// TIA Portal V16 export
// export: Created 2021-07-21T13:08:43.8324365Z, ExportSetting WithDefaults, DisplayName Totally Integrated Automation Portal, DisplayVersion V16 Update 3, DisplayName TIA Portal Version Control Interface, DisplayVersion V16 Update 2, DisplayName TIA Portal Openness, DisplayVersion V16 Update 3, DisplayName STEP 7 Professional, DisplayVersion V16 Update 3, DisplayName STEP 7 Safety, DisplayVersion V16, DisplayName WinCC Professional, DisplayVersion V16 Update 3
TYPE "UT31001_Dy_DevValveIsol"
TITLE = Dynamic UDT [Instrumentation] — Analog Instrument Read, Scale and Monitor
// Analogue Instrument Read and Scale
// stored: IsFailsafeCompliant false
   STRUCT
      revInfo : "UT01000_St_SysRevision";   // Revision information
      ___________0010_0 { ExternalAccessible := 'False'; ExternalVisible := 'False'; ExternalWritable := 'False'} : Int;
      ___________0010_1 { ExternalAccessible := 'False'; ExternalVisible := 'False'; ExternalWritable := 'False'} : Int;   // ▀▀▀▀ STATUS (FOR BLOCK ICON AND SYMBOL)
      status_Closed : Bool;   // STATUS — Valve is confirmed closed (1 = valve is closed, 0 = valve is not closed)
      status_Open : Bool;   // STATUS — Valve is confirmed open (1 = valve is open, 0 = valve is not open)
      status_Closing : Bool;   // STATUS — Valve is closing (1 = valve is closing, 0 = valve is not closing)
      status_Opening : Bool;   // STATUS — Valve is opening (1 = valve is opening, 0 = valve is not opening)
      status_Operating : Bool;   // STATUS — Valve is changing state (1 = valve is opening or closing, 0 = valve is not moving)
      status_Fault : Bool;   // STATUS — Valve is in fault (1 = fault present, 0 = healthy)
      status_Energised : Bool;   // STATUS — Valve output is on (1 = valve energised, 0 = valve deenergised)
      status_Aut : Bool;   // STATUS — Automatic mode active (1 = in automatic mode, 0 = not in automatic mode)
      status_Man : Bool;   // STATUS — Manual mode active (1 = in manual mode, 0 = not in manual mode)
      status_EStop : Bool;   // STATUS — E_STOP safety signal is active (1 = E_STOP active, 0 = E_STOP not active)
      status_Trip : Bool;   // STATUS — TRIP signal is active (1 = TRIP active, 0 = TRIP not active)
      status_Ilock : Bool;   // STATUS — INTERLOCK signal is active (1 = INTERLOCK active, 0 = INTERLOCK not active)
      status_Perm : Bool;   // STATUS — PERMISSIVE signal is active (1 = PERMISSIVE active, 0 = PERMISSIVE not active)
      status_BypassOn : Bool;   // STATUS — Valve is in bypass mode (1 = bypass mode on, 0 = normal)
      status_SimOn : Bool;   // STATUS — Valve is in simulation mode (1 = simulation mode on, 0 = normal)
      status_RemoteOn : Bool;   // STATUS — Valve is in remote mode (1 = remote mode, 0 = remote mode off)
      status_LocalOn : Bool;   // STATUS — Valve is in local mode (1 = local mode, 0 = local mode off)
      status_RLOff : Bool;   // STATUS — Remote/local mode disabled (1 = ALL mode on, 0 = RL mode selected)
      ___________0020_0 { ExternalAccessible := 'False'; ExternalVisible := 'False'; ExternalWritable := 'False'} : Int;
      ___________0020_1 { ExternalAccessible := 'False'; ExternalVisible := 'False'; ExternalWritable := 'False'} : Int;   // ▀▀▀▀ MESSAGES (ALARMS, WARNINGS, FAULTS AND EVENTS)
      msg_FailToOpen : Bool;   // MESSAGE — Alarm – “Fail to open” is active (1 = alarm active, 0 = alarm not active)
      msg_FailToClose : Bool;   // MESSAGE — Alarm – “Fail to close” is active (1 = alarm active, 0 = alarm not active)
      msg_FailWhileOpen : Bool;   // MESSAGE — Alarm – “Fail while open” is active (1 = alarm active, 0 = alarm not active)
      msg_FailWhileClosed : Bool;   // MESSAGE — Alarm – “Fail while closed” is active (1 = alarm active, 0 = alarm not active)
      msg_Flt_External : Bool;   // MESSAGE — Alarm – “External fault” is active (1 = alarm active, 0 = alarm not active)
      ___________0030_0 { ExternalAccessible := 'False'; ExternalVisible := 'False'; ExternalWritable := 'False'} : Int;
      ___________0030_1 { ExternalAccessible := 'False'; ExternalVisible := 'False'; ExternalWritable := 'False'} : Int;   // ▀▀▀▀ OPERATING MODE SELECTION (FROM FACEPLATE OR PANEL)
      mode_AutMan : Bool;   // MODE — Automatic or manual mode selection (1 = automatic mode, 0 = manual mode)
      mode_BypassOn : Bool;   // MODE — Bypass mode (1 = bypass mode active, 0 = normal)
      mode_SimOn : Bool;   // MODE — Simulation mode (1 = simulation mode active, 0 = normal)
      mode_SimValue : Int;   // MODE — Simulation value (0 no limits, 1 always open, 2 always closed, 3 follow demand)
      mode_RemoteOn : Bool;   // MODE — Local HMI control enabled (1 = control active, 0 = control disabled or N/A)
      mode_LocalOn : Bool;   // MODE — Remote SCADA control enabled (1 = control active, 0 = control disabled or N/A)
      mode_Reset : Bool;   // MODE — Fault reset (1 = Reset any faults – 1 cycle only, 0 = does nothing)
      ___________0040_0 { ExternalAccessible := 'False'; ExternalVisible := 'False'; ExternalWritable := 'False'} : Int;
      ___________0040_1 { ExternalAccessible := 'False'; ExternalVisible := 'False'; ExternalWritable := 'False'} : Int;   // ▀▀▀▀ CONTROL SIGNALS (TO OPERATE THE DEVICE)
      ctrl_Aut_OpenClose : Bool;   // CONTROL — Auto mode open or close valve (1 = open valve in auto, 0 = close valve in auto)
      ctrl_Man_OpenClose : Bool;   // CONTROL — Manual mode open or close valve (1 = open valve in man, 0 = close valve in man)
      ___________0050_0 { ExternalAccessible := 'False'; ExternalVisible := 'False'; ExternalWritable := 'False'} : Int;
      ___________0050_1 { ExternalAccessible := 'False'; ExternalVisible := 'False'; ExternalWritable := 'False'} : Int;   // ▀▀▀▀ BATCH AND BOOKING DATA
      batch_ID : Int;   // BATCH — Booking ID (optional for batch operations)
      ___________0060_0 { ExternalAccessible := 'False'; ExternalVisible := 'False'; ExternalWritable := 'False'} : Int;
      ___________0060_1 { ExternalAccessible := 'False'; ExternalVisible := 'False'; ExternalWritable := 'False'} : Int;   // ▀▀▀▀ LIVE DATA (SCALED READING & TIMER VALUES)
      actual_Operating_Timer : Real;   // ACTUAL — Timer value — operating opening/closing timer actual value [seconds]
      ___________0090_0 { ExternalAccessible := 'False'; ExternalVisible := 'False'; ExternalWritable := 'False'} : Int;
      ___________0090_1 { ExternalAccessible := 'False'; ExternalVisible := 'False'; ExternalWritable := 'False'} : Int;   // ▀▀▀▀ BLOCK INTERNAL WORKING AND STORAGE AREA
      "$derived_fbk_open" : Bool;   // INTERNAL — Derived feedback open signal (if CONFIG_FBK_OPEN_EN = 0)
      "$derived_fbk_closed" : Bool;   // INTERNAL — Derived feedback closed signal (if CONFIG_FBK_CLOSED_EN = 0)
      "$sim_fbk_open" : Bool;   // INTERNAL — Simulated feedback open signal (if mode_SimOn = 1)
      "$sim_fbk_closed" : Bool;   // INTERNAL — Simulated feedback closed signal (if mode_SimOn = 1)
      "$ctrl_OpenClose" : Bool;   // INTERNAL — actual open or close control signal passed to the valve (1 = open, 0 = close)
      "$pret_Open" : Bool;   // INTERNAL — Edge retention (+ve) rising edge of ctrl_OpenClose (change of state to open)
      "$nret_Close" : Bool;   // INTERNAL — Edge retention (-ve) falling edge of ctrl_OpenClose (change of state to close)
   END_STRUCT;
   // revInfo.REV_BLOCK := 'UT31001';
   // revInfo.REV_NUMBER := '000.102';
   // revInfo.REV_DATE := '2021-07-21';
   // revInfo.REV_AUTHOR := 'M. Gledhill';
END_TYPE
